FUNCTION_BLOCK Device_PartSensor

VAR_INPUT
	iSensor1On AT %I* 	: BOOL;
END_VAR

VAR_OUTPUT
	oPartPresent		: BOOL;
END_VAR

VAR_INPUT PERSISTENT
	Name				: STRING;
	
	cOnDelay 			: TIME;
	cOffDelay 			: TIME;
END_VAR

VAR
	OnDelayTimer 		: TON;
	OffDelayTimer 		: TOF;
	SetReset: SR;
END_VAR

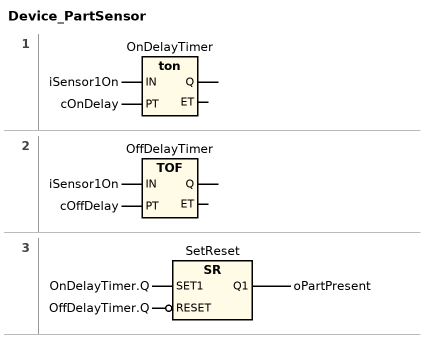
// NETWORK 1
OnDelayTimer(IN := iSensor1On, PT := cOnDelay); // ton

// NETWORK 2
OffDelayTimer(IN := iSensor1On, PT := cOffDelay); // TOF

// NETWORK 3
SetReset(SET1 := OnDelayTimer.Q, RESET := NOT OffDelayTimer.Q); // SR
oPartPresent := SetReset.Q1;

END_FUNCTION_BLOCK

(* stored: Version 1.1.0.1, ProductVersion 3.1.4022.11
   POU Device_PartSensor: Id {4f6ddd2d-9034-48b3-92a3-4056cd68e165}, SpecialFunc None *)
